FUNCTION_BLOCK Transport (* Basic Function Block Type *)
  (* Standard: 61499-2 *)
  (* Version 0.0, 2015-03-24, 4DIAC-IDE, 4DIAC-Consortium *)
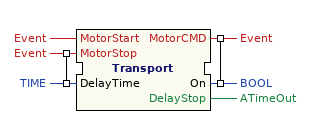
  EVENT_INPUT
    MotorStart; (* Start the conveyor belt *)
    MotorStop WITH DelayTime; (* Stop the conveyor belt *)
  END_EVENT
  EVENT_OUTPUT
    MotorCMD WITH On; (* Send motor command *)
  END_EVENT
  VAR_INPUT
    DelayTime : TIME;
  END_VAR
  VAR_OUTPUT
    On : BOOL; (* Motor control output *)
  END_VAR
  PLUGS
    DelayStop : ATimeOut;
  END_PLUGS
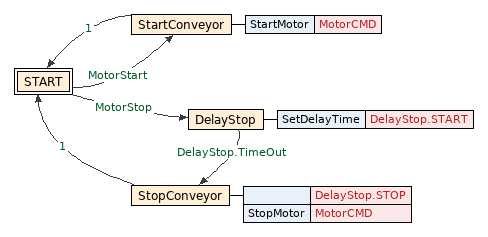
  EC_STATES
    START; (* Initial State *)
    StartConveyor : StartMotor -> MotorCMD; (* Initialization *)
    StopConveyor : -> DelayStop.STOP, StopMotor -> MotorCMD;
    DelayStop : SetDelayTime -> DelayStop.START;
  END_STATES
  EC_TRANSITIONS
    START TO StartConveyor := MotorStart;
    StopConveyor TO START := 1;
    StartConveyor TO START := 1;
    START TO DelayStop := MotorStop;
    DelayStop TO StopConveyor := DelayStop.TimeOut;
  END_TRANSITIONS
  ALGORITHM StartMotor IN ST: (* Start motor *)
On := TRUE;
  END_ALGORITHM
  ALGORITHM StopMotor IN ST: (* Stop motor *)
On := FALSE;
  END_ALGORITHM
  ALGORITHM SetDelayTime IN ST: (* new algorithm *)
DelayStop.DT :=DelayTime;
  END_ALGORITHM
  SERVICE transport_interface/transport_implementation (* Basic Function Block Type *)
    SEQUENCE StartConveyor
      transport_interface.MotorStart() -> transport_interface.MotorCMD(On = true);
    END_SEQUENCE
    SEQUENCE DelayStop
      transport_interface.MotorStop() -> transport_interface.DelayStop.START(DelayStop.DT =DelayTime);
      transport_interface.DelayStop.TimeOut() -> transport_interface.DelayStop.STOP() -> transport_interface.MotorCMD(On = false);
    END_SEQUENCE
  END_SERVICE
END_FUNCTION_BLOCK
